// TIA Portal V20 export
FUNCTION_BLOCK "FB_Counter"   // FB40, SCL
{ S7_Optimized_Access := 'TRUE' }
// stored: MemoryReserve 100, SetENOAutomatically false
   VAR_INPUT
      iIncrement : Bool;
      iReset : Bool;
      iLimit : UDInt;
   END_VAR
   VAR_OUTPUT
      oLimitReached : Bool;
   END_VAR
   VAR
      sRT_Increment { ExternalAccessible := 'False'; ExternalVisible := 'False'; ExternalWritable := 'False'} : R_TRIG;
      sCounter { S7_SetPoint := 'True'} : UDInt;
      sCounterNoReset : UDInt;
   END_VAR
BEGIN
   REGION Description header 
       //==================================================================================
       // POSALUX Swiss SA / (C) Copyright 2025
       //----------------------------------------------------------------------------------
       // Title: FB_Counter
       // Comment/Function: This function allows:
       //                      - Counting Pulse
       //
       // Author: Fabien Waldt
       // Engineering: TIA Portal v19
       //----------------------------------------------------------------------------------
       // Change log table:
       // Version  | Date     | Expert in charge | Changes applied
       // ---------|----------|------------------|------------------------------------
       // 00.00.01 | 20250718 | WFA              | First released version
       // ==================================================================================
   END_REGION

   REGION Counter Reset
       IF #iReset THEN
           #sCounter := 0;
       END_IF;

       IF #sCounterNoReset >= 4294967295 THEN
           #sCounterNoReset := 0;
       END_IF;
   END_REGION

   REGION Counter Increment
       #sRT_Increment(CLK := #iIncrement);

       IF #sRT_Increment.Q THEN
           #sCounter := #sCounter + 1;
           #sCounterNoReset := #sCounterNoReset + 1;
       END_IF;
   END_REGION ;

   REGION Limit Reached
       #oLimitReached := #sCounter >= #iLimit;
   END_REGION ;
END_FUNCTION_BLOCK
